// Mitsubishi GX Works2 project: TestCLPunching   PLC: FX3U/FX3UC

TYPE ST_ServoMotorInterface : STRUCT
  bBusy : BOOL;
  bError : BOOL;
  bDone : BOOL;
  bServoEnabled : BOOL;
  bEnable : BOOL;
  bStop : BOOL;
  bAbort : BOOL;
  bReset : BOOL;
  bJogPos : BOOL;
  bJogNeg : BOOL;
  bMoveRel : BOOL;
  rMoveDist : REAL;
  iMoveVel : DINT;
  iMoveAccel : DINT;
  iOutChannel : INT;
  iRevChannel : INT;
  iMoveDelay : WORD;
END_STRUCT END_TYPE

TYPE ST_1SolCylinderInterface : STRUCT
  bBusy : BOOL;
  bError : BOOL;
  bDone : BOOL;
  bGoActive : BOOL;
  bReset : BOOL;
  tDelayTime : TIME;
  tTimeout : TIME;
END_STRUCT END_TYPE

// global labels: Global1
VAR_GLOBAL
  objServoMotor : CL_ServoMotor;
  biServoINP AT X005 : BOOL;
  biServoRD AT X006 : BOOL;
  biServoALM AT X007 : BOOL;
  boServoSON AT Y004 : BOOL;
  boServoRES AT Y005 : BOOL;
  boServoEM2 AT Y003 : BOOL;
  stServoMotor AT Detail Setting : ST_ServoMotorInterface;
  tboxPulsePerRev AT D200 : DINT;
  tboxRadius AT D202 : REAL;
  tboxMoveVel AT D204 : DINT;
  tboxMoveAccel AT D206 : DINT;
  tboxMoveDist AT D124 : REAL;
  bCommandComplete AT M8029 : BOOL;
END_VAR
VAR_GLOBAL CONSTANT
  iOutChannel1 : INT;
  iRevChannel1 : INT := 1;
  iMoveDelay1 : WORD := 100;
END_VAR
VAR_GLOBAL
  boServoNPz AT Y001 : BOOL;
  objPunching : CL_1Sol1SenCylinder;
  stPunching AT Detail Setting : ST_1SolCylinderInterface;
  biPunchingDone AT X002 : BOOL;
  boPunchingOutput AT Y006 : BOOL;
  tboxPunchingDelayTime AT D210 : DINT;
  tboxPunchingTimeout AT D212 : DINT;
  bPunchingDone : BOOL;
END_VAR

// task Task_01 (event TRUE, interval 0, priority 31): POU_01

PROGRAM POU_01
objServoMotor(biINP := biServoINP,
								biRD := biServoRD,
								biALM := biServoALM,
								boNPz := boServoNPz,
								boEM2 := boServoEM2,
								boRES := boServoRES,
								boSON := boServoSON,
								
								bEnable := stServoMotor.bEnable,
								bStop := stServoMotor.bStop,
								bAbort := stServoMotor.bAbort,
								bReset := stServoMotor.bReset,
								iOutChannel := stServoMotor.iOutChannel,
								iRevChannel := stServoMotor.iRevChannel,
								iMoveDelay := stServoMotor.iMoveDelay,
								iPulsePerRev := tboxPulsePerRev,
								rRadius := tboxRadius,
								
								bJogPos := stServoMotor.bJogPos,
								bJogNeg := stServoMotor.bJogNeg,
								
								bMoveRel := stServoMotor.bMoveRel,
								rMoveDist := stServoMotor.rMoveDist,
								iMoveVel := tboxMoveVel,
								iMoveAccel := tboxMoveAccel,

								bBusy := stServoMotor.bBusy,
								bDone := stServoMotor.bDone,
								bError := stServoMotor.bError,
								bServoEnabled := stServoMotor.bServoEnabled);

objPunching(biSensorDone := bPunchingDone,
							biActiveFeedback := boPunchingOutput,
							boSolenoid := boPunchingOutput,
							
							bGoActive := stPunching.bGoActive,
							bReset := stPunching.bReset,
							tDelayTime := tboxPunchingDelayTime,
							tTimeout := tboxPunchingTimeout,

							bBusy := stPunching.bBusy,
							bInHomePos := stPunching.bDone,
							bError := stPunching.bError);
END_PROGRAM

FUNCTION_BLOCK CL_ServoMotor
VAR_INPUT
  biINP : BOOL;
  biRD : BOOL;
  biALM : BOOL;
  bEnable : BOOL;
  bStop : BOOL;
  bAbort : BOOL;
  bReset : BOOL;
  bJogPos : BOOL;
  bJogNeg : BOOL;
  bMoveRel : BOOL;
  rMoveDist : REAL;
END_VAR
VAR_OUTPUT
  boEM2 : BOOL;
  boSON : BOOL;
  boRES : BOOL;
  bBusy : BOOL;
  bError : BOOL;
  bDone : BOOL;
  bServoEnabled : BOOL;
END_VAR
VAR
  iState : INT;
  fbResetHold : TP_10;
  bResetHold : BOOL;
  fbMoveDelay : TON;
END_VAR
VAR_INPUT
  iMoveDelay : WORD;
END_VAR
VAR
  tMoveDelay : TIME;
  iStopState : INT;
END_VAR
VAR_INPUT
  iMoveVel : DINT;
  iMoveAccel : DINT;
  iPulsePerRev : DINT;
  rRadius : REAL;
END_VAR
VAR
  iFrequency : DINT;
  iPulse : DINT;
  iAccel : DINT;
  bOutPulse : BOOL;
END_VAR
VAR_INPUT
  iOutChannel : INT;
  iRevChannel : INT;
END_VAR
VAR
  bInCommand : BOOL;
  bCompleted : BOOL;
  tonDelayComplete : TON_10;
  bCompletedHold : BOOL;
  bDebug : BOOL;
END_VAR
VAR_OUTPUT
  boNPz : BOOL;
END_VAR
(*Main State Machine*)
CASE iState OF 
		0: 	(*Unenabled, wait for Enable command*)
				IF bEnable AND NOT bStop AND NOT bError THEN
						iState := 10;
				END_IF;
				
		10: 	(*Servo On*)
				IF bServoEnabled THEN
						iState := 20;
				END_IF;
						
		20: 	(*Servo Ready, wait for moving command*)
				IF bJogPos AND NOT bStop AND NOT bError THEN
						iState := 100;
				ELSIF bJogNeg AND NOT bStop AND NOT bError THEN
						iState := 140;
				ELSIF bMoveRel AND NOT bStop AND NOT bError THEN
						iState := 200;
				END_IF;
				
		100: 	(*Calculate number of pulse*)			
				iFrequency := 50000;
				iPulse := REAL_TO_DINT(DINT_TO_REAL(iPulsePerRev)*1000.0/(2.0*3.1415926*rRadius));
				iAccel := iMoveAccel;
				iState := 110;
				
		110: 	(*Execute Jog Pos command*)
				IF NOT bJogPos THEN 
						iState := 20;
				END_IF;
				
		140: 	(*Calculate number of pulse*)			
				iFrequency := 50000;
				iPulse := REAL_TO_DINT(DINT_TO_REAL(iPulsePerRev)*1000.0/(2.0*3.1415926*rRadius));
				iAccel := iMoveAccel;
				iState := 150;
				
		150: 	(*Execute Jog Neg command*)
				IF NOT bJogNeg THEN
						iState := 20;
				END_IF;
				
		200: 	(*Calculate number of pulse*)
				iFrequency := REAL_TO_DINT(DINT_TO_REAL(iPulsePerRev*iMoveVel)/60.0);
				iPulse := REAL_TO_DINT(DINT_TO_REAL(iPulsePerRev)*rMoveDist/(2.0*3.1415926*rRadius));	
				iAccel := iMoveAccel;
				tMoveDelay := WORD_TO_TIME(iMoveDelay);
				iState := 210;
		
		210: 	(*Execute Move Relative command*)
				IF tonDelayComplete.Q AND fbMoveDelay.Q THEN		
						iState := 220;
				END_IF;		
				
		220: 	(*Move Relative done, wait for command release*)
				IF NOT bMoveRel THEN
						iState := 20;
				END_IF;
				
END_CASE;
	
(*Procedure*)
		(*Abort*)
		IF bAbort OR NOT bEnable OR bError THEN
				iState := 0;
				iStopState := 0;
		END_IF;
		
		(*Reset*)
		IF bReset AND bError THEN
				iState := 0;
				iStopState := 0;
		END_IF;		
		
		(*Stop*)
		CASE iStopState OF
				0: 	(*Wait for stop signal*)
						IF bStop THEN
								iStopState := 10;
						END_IF;
						
				10: 	(*Execute Stop*)
						IF iState > 20 THEN
								iState := 20;
						END_IF;
						IF biINP THEN
								iStopState := 20;
						END_IF;
						
				20: 	(*Stop done, wait for command release*)
						IF NOT bStop THEN
								iStopState := 0;
						END_IF;
		END_CASE;	

(*State Action*)
		boSON := (iState >= 10);																			(*Enable Servo Motor*)	
		boEM2 := NOT bAbort AND biALM;													(*Abort Servo Motor*)
		boRES := fbResetHold.Q AND NOT biALM;									(*Reset Servo Motor*)		
		
		bBusy := (iState = 110) OR (iState = 150) OR (iState = 210) OR (iStopState = 10);
		bDone := (iState = 220) OR (iStopState = 20);									(*Servo movement is done*)
		bServoEnabled := biRD;																		(*Servo is powered on*)
	
		SET(NOT biALM, bError);																		(*Notify Servo Motor Error*)
		RST((bReset AND bError), bError);													(*Reset object error*)	
		
		bInCommand:= ((iState = 110) OR (iState = 150) OR (iState = 210)) AND NOT (iStopState = 10);	(*Enable Pulse*)
		boNPz := ((iState = 150) OR (rMoveDist < 0.0));												(*Reverse rotation*)
		
		SET(bCompleted, bCompletedHold);
		RST(NOT (iState = 210), bCompletedHold);
		bResetHold := (bReset AND NOT fbResetHold.Q) OR (bResetHold AND fbResetHold.Q) ;
	
(*Function Block Call*)
fbResetHold(IN := bResetHold, PT := t#600ms);
fbMoveDelay(IN := bMoveRel AND bServoEnabled AND NOT bStop AND NOT bAbort AND NOT bError, PT := tMoveDelay);
tonDelayComplete(IN := biINP AND bCompletedHold, PT:= t#50ms);

(*Output pulse to server drive*)
bOutPulse := (LDP(TRUE, bInCommand) OR bOutPulse) AND NOT (bCompleted AND bMoveRel) AND NOT LDF(TRUE, bInCommand);		(*Output pulse command*)

CASE iOutChannel OF 
	0: 	(*Y000*)
			DPLSR(bOutPulse, iFrequency, iPulse, iAccel, Y000);
			bDebug := M8013;
	1:		(*Y001*)
			DPLSR(bOutPulse, iFrequency, iPulse, iAccel, Y001);
	2:		(*Y002*)
			DPLSR(bOutPulse, iFrequency, iPulse, iAccel, Y002);
END_CASE;
bCompleted := bCommandComplete;
END_FUNCTION_BLOCK

FUNCTION_BLOCK CL_1Sol1SenCylinder
VAR_INPUT
  biSensorDone : BOOL;
  bGoActive : BOOL;
  bReset : BOOL;
END_VAR
VAR_OUTPUT
  boSolenoid : BOOL;
  bBusy : BOOL;
  bInHomePos : BOOL;
  bError : BOOL;
END_VAR
VAR_INPUT
  tDelayTime : DINT;
  tTimeout : DINT;
END_VAR
VAR
  fbDelayTime : TON;
  fbTimeout : TON;
END_VAR
VAR_INPUT
  biActiveFeedback : BOOL;
END_VAR
VAR
  bSensorDoneHold : BOOL;
  bBusyPulse : BOOL;
  tDelay : TIME;
  tTimeoutz : TIME;
END_VAR
(*Activate Output: Enable solenoid on valve*) 
boSolenoid := LDP(TRUE, bGoActive) OR boSolenoid AND NOT fbTimeout.Q AND NOT biSensorDone;

(*Process Input: Wait for sensors signal*)
SET(biSensorDone, bSensorDoneHold);
RST(LDP(TRUE, bBusy), bSensorDoneHold);
bInHomePos := fbDelayTime.Q AND bSensorDoneHold;
bBusy := biActiveFeedback AND NOT biSensorDone;

(*Error handling*)
		(*Notify timeout error*)
		SET(fbTimeout.Q, bError);

		(*Reset timeout error*)
		RST(bReset, bError);

(*Timers call*)
tDelay := DINT_TO_TIME(tDelayTime);
tTimeoutz := DINT_TO_TIME(tTimeout);
fbDelayTime(IN := NOT bBusy, PT := tDelay );
fbTimeout(IN := bBusy, PT := tTimeoutz );
END_FUNCTION_BLOCK
